// TwinCAT 3 PLC project ScopeTestPLC
// ProgramVersion: 3.1.4024.0
// libraries:
//   Tc2_MC2, * (Beckhoff Automation GmbH)
//   Tc2_Standard, * (Beckhoff Automation GmbH)
//   Tc2_System, * (Beckhoff Automation GmbH)
//   Tc3_Module, * (Beckhoff Automation GmbH)
// project tree:
//   DUTs/ EAxisCycleStates.TcDUT
//   GVLs/ Axes.TcGVL (not stored)
//   / PlcTask.TcTTO
//   POUs/ MAIN.TcPOU, MoveVirtualAxis.TcPOU
// real-time tasks:
//   TASK PlcTask: cycle T#10ms, priority 20, ADS port 350
// motion (NC):
// variable links:
//   ScopeTestPLC Instance <-> NC-Task 1 SAF/Axes/Axis 1
//     PlcTask Inputs/Axes.Axis1.NcToPlc <-> Outputs/ToPlc
//     PlcTask Outputs/Axes.Axis1.PlcToNc <-> Inputs/FromPlc

CONFIGURATION ScopeTestPLC
    RESOURCE PLC ON TwinCAT3
        TASK PlcTask(INTERVAL := T#10ms, PRIORITY := 20);
        PROGRAM MAIN WITH PlcTask : MAIN;
    END_RESOURCE
END_CONFIGURATION

// ---- DUTs/EAxisCycleStates.TcDUT
{attribute 'qualified_only'}
{attribute 'strict'}
TYPE EAxisCycleStates :
(
    Init := 0,           // Inicialização
    MovingTo1000 := 1,   // Movendo para a posição 1000
    WaitingAt1000 := 2,  // Aguardando por 3 segundos na posição 1000
    MovingTo0 := 3,      // Movendo para a posição 0
    WaitingAt0 := 4,     // Aguardando por 3 segundos na posição 0
    Stop := 5            // Estado de parada (desativado)
); 
END_TYPE

// ---- POUs/MAIN.TcPOU
PROGRAM MAIN
VAR
	MaquinaLigada: BOOL;
	bHabilita: BOOL;
	fb_Habilita1: MC_Power;
END_VAR

//Ler Status
	Axes.Axis1.ReadStatus();
	
//Habilitar Eixo1
	IF MaquinaLigada THEN
		bHabilita := 1;
	ELSE
		bHabilita := 0;
	END_IF
	fb_Habilita1(
		Axis:= Axes.Axis1, 
		Enable:= bHabilita, 
		Enable_Positive:= bHabilita, 
		Enable_Negative:= bHabilita, 
		Override:= 100.0);

//Chama o programa de movimento

END_PROGRAM

// ---- POUs/MoveVirtualAxis.TcPOU
PROGRAM MoveVirtualAxis
VAR
    currentState : EAxisCycleStates := EAxisCycleStates.Init; // Estado inicial
    nextState : EAxisCycleStates;                        // Próximo estado

    // Variáveis de controle
    axisPosition : LREAL;     					// Posição do eixo virtual
    targetPosition : REAL; 						// Posição alvo
	Timer: TON;
	isCycleActive : BOOL := TRUE;   // Indicador de ciclo ativo (ligado/desligado pelo usuário)
	fb_MoveAbsolutoEixo1: MC_MoveAbsolute;
	fb_MoveAbsolutoEixo2: MC_MoveAbsolute;
	bMoverEixo1Abs: BOOL;
	bMoverEixo1Abs2: BOOL;
END_VAR


CASE currentState OF
    EAxisCycleStates.Init:
        // Inicializa o sistema e define a posição alvo como 1000
        axisPosition := Axes.Axis1.NcToPlc.ActPos;
        targetPosition := 1000.0;
        nextState := EAxisCycleStates.MovingTo1000; // Vai mover para a posição 1000
		//Move Absolute
	
        
    EAxisCycleStates.MovingTo1000:
        // Movendo o eixo para a posição 1000
        IF axisPosition < targetPosition THEN
            fb_MoveAbsolutoEixo1(
				Axis:= Axes.Axis1, 
				Execute:= bMoverEixo1Abs, 
				Position:= targetPosition, 
				Velocity:= 500.0); // Atualiza a posição
        ELSE
            // Quando atingir a posição 1000, inicia o temporizador de 3 segundos
            Timer(IN:= TRUE, PT:= T#3S);
            nextState := EAxisCycleStates.WaitingAt1000;
        END_IF
        
    EAxisCycleStates.WaitingAt1000:
        // Espera 3 segundos na posição 1000
        IF Timer.Q THEN
            targetPosition := 0.0;    // Define a próxima posição como 0
            Timer(IN := FALSE);       // Reseta o temporizador
            nextState := EAxisCycleStates.MovingTo0; // Muda para mover de volta para 0
			bMoverEixo1Abs := FALSE;
			bMoverEixo1Abs2 := TRUE;
        END_IF

    EAxisCycleStates.MovingTo0:
        // Movendo o eixo para a posição 0
        IF axisPosition > targetPosition THEN
            fb_MoveAbsolutoEixo2(
				Axis:= Axes.Axis1, 
				Execute:= bMoverEixo1Abs2, 
				Position:= 0, 
				Velocity:= 500.0);; // Atualiza a posição
        ELSE
            // Quando atingir a posição 0, inicia o temporizador de 3 segundos
            Timer(IN := TRUE, PT := T#3S);
            nextState := EAxisCycleStates.WaitingAt0;
        END_IF
        
    EAxisCycleStates.WaitingAt0:
        // Espera 3 segundos na posição 0
        IF Timer.Q THEN
            targetPosition := 1000.0; // Define a próxima posição como 1000
            Timer(IN := FALSE);       // Reseta o temporizador
            nextState := EAxisCycleStates.MovingTo1000; // Muda para mover de volta para 1000
			bMoverEixo1Abs := TRUE;
			bMoverEixo1Abs2 := FALSE;
        END_IF
        
END_CASE


// Transição de estados
currentState := nextState;

END_PROGRAM
